// TwinCAT 3 PLC project ControlPanel
// ProgramVersion: 3.1.4024.0
// libraries:
//   Tc2_HVAC, * (Beckhoff Automation GmbH)
//   Tc2_ModbusSrv, * (Beckhoff Automation GmbH)
//   Tc2_Standard, * (Beckhoff Automation GmbH)
//   Tc2_System, * (Beckhoff Automation GmbH)
//   Tc3_Module, * (Beckhoff Automation GmbH)
// project tree:
//   DUTs/ FactoryIO_Input.TcDUT, FactoryIO_Output.TcDUT
//   GVLs/ GVL.TcGVL, GVL_System.TcGVL
//   / PlcTask.TcTTO
//   POUs/ Blink.TcPOU, ControlPanel.TcPOU, MAIN.TcPOU, MyBlink.TcPOU, ReadModbusCoils.TcPOU, ReadModbusReg.TcPOU
// real-time tasks:
//   TASK PlcTask: cycle T#10ms, priority 20, ADS port 350

CONFIGURATION ControlPanel
    RESOURCE PLC ON TwinCAT3
        TASK PlcTask(INTERVAL := T#10ms, PRIORITY := 20);
        PROGRAM MAIN WITH PlcTask : MAIN;
    END_RESOURCE
END_CONFIGURATION

// ---- DUTs/FactoryIO_Input.TcDUT
TYPE FactoryIO_Input :
STRUCT
	bAtBufferEntry	:	BOOL;
	bAtBufferExit	:	BOOL;
	bAtExit			:	BOOL;
	bStartButton	: 	BOOL;
	bResetButton	: 	BOOL;
	bStopButton		: 	BOOL;
	bAuto			: 	BOOL;
	bEmgStop		: 	BOOL;
	bManual			: 	BOOL;
	nSpeed			:	WORD;
END_STRUCT
END_TYPE

// ---- DUTs/FactoryIO_Output.TcDUT
TYPE FactoryIO_Output :
STRUCT
	bStopBlade		:	BOOL;
	bStartLight		:	BOOL;
	bResetLight		:	BOOL;
	bStopLight		:	BOOL;
	nBufferConveyor	: 	WORD;
	nExitConveyor	: 	WORD;
	nCounter		:	WORD;
END_STRUCT
END_TYPE

// ---- GVLs/GVL.TcGVL
{attribute 'qualified_only'}
VAR_GLOBAL
	// Digital IO in FactoryIO Outputs
	mb_Input_Coils		:	ARRAY [0..3] OF BOOL;
	// Digital IO in FactoryIO Inputs
	mb_Output_Coils		:   ARRAY [0..9] OF BOOL;
	// Analog IO in FactoryIO Outputs
	mb_Input_Registers	: 	ARRAY [0..2] OF WORD;
	// Analog IO in FactoryIO Inputs
	mb_Output_Registers	: 	ARRAY [0..1] OF WORD;
	
	nState				: INT;
END_VAR

// ---- GVLs/GVL_System.TcGVL
{attribute 'qualified_only'}
VAR_GLOBAL
	isResetON	: BOOL;
	isStopON	: BOOL;
	isEmgStopON	: BOOL;
	
END_VAR

// ---- POUs/MAIN.TcPOU
PROGRAM MAIN
VAR
	(*
	fbReadRegs        : FB_MBReadRegs;
    bReadRegs         : BOOL;
    bReadRegsBusy     : BOOL;
    bReadRegsError    : BOOL;
    nReadRegsErrorId  : UDINT;
    nReadRegsCount    : UDINT;
    nQuantity         : WORD:=2;
    nMBAddr           : WORD:=24;
    arrData           : ARRAY [1..2] OF WORD;
	*)
	
	//myBlink	: Array[0..7] OF MyBlink();
	redBlink	: MyBlink();
	yellowBlink	: MyBlink();
	greenBlink	: MyBlink();
	controlPanel 	:	ControlPanel();
	
END_VAR

Blink();


ControlPanel();

END_PROGRAM

// ---- POUs/MyBlink.TcPOU
FUNCTION_BLOCK MyBlink
VAR_INPUT
	tBlinkTime			: TON;
	bEnable				: BOOL;
	bBlinkHz			: BOOL;
	tTimeOn				: TIME := T#2S;
	tTimeOff 			: TIME := tTimeOn/2;
END_VAR
VAR_OUTPUT
	bBlink				: BOOL;
END_VAR
VAR
END_VAR

// SET Timer ON
tBlinkTime(IN:=NOT tBlinkTime.Q, PT:= tTimeON);

// Set Timer OFF
bBlinkHz := tBlinkTime.ET >= tTimeOff;

// OUTPUT
bBlink := bBlinkHz AND bEnable;

END_FUNCTION_BLOCK

// ---- POUs/ControlPanel.TcPOU
FUNCTION_BLOCK ControlPanel
VAR_INPUT
	
	
END_VAR
VAR_OUTPUT
	
END_VAR
VAR
	isResetON	: BOOL;
	isStopON	: BOOL;
	isEmgStopON	: BOOL;
	isSystemON	: BOOL;
	
	factoryIO_Input	: FactoryIO_Input;
	i	: INT;
	
	(*
	bAtBufferEntry	:	BOOL;
	bAtBufferExit	:	BOOL;
	bAtExit			:	BOOL;
	bStartButton	: 	BOOL;
	bResetButton	: 	BOOL;
	bStopButton		: 	BOOL;
	bAuto			: 	BOOL;
	bEmgStop		: 	BOOL;
	bManual			: 	BOOL;
	*)
	
	blink			: MyBlink();
END_VAR

{region "READ Values from Sensors"}
	(*
	bAtBufferEntry	:=	GVL.mb_Output_Coils[0];
	bAtBufferExit	:= 	GVL.mb_Output_Coils[1];
	bAtExit			:=	GVL.mb_Output_Coils[2];
	bStartButton	:=	GVL.mb_Output_Coils[3];
	bResetButton	:= 	GVL.mb_Output_Coils[4];
	bStopButton		:= 	GVL.mb_Output_Coils[5];
	bAuto			:=	GVL.mb_Output_Coils[6];
	bEmgStop	 	:= 	GVL.mb_Output_Coils[7];
	bManual	 		:= 	GVL.mb_Output_Coils[8];
	*)
	 
	factoryIO_Input.bAtBufferEntry	:=	GVL.mb_Output_Coils[0];
	factoryIO_Input.bAtBufferExit	:=	GVL.mb_Output_Coils[1];
	factoryIO_Input.bAtExit			:=	GVL.mb_Output_Coils[2];
	factoryIO_Input.bStartButton	:=	GVL.mb_Output_Coils[3];
	factoryIO_Input.bResetButton	:=	GVL.mb_Output_Coils[4];
	factoryIO_Input.bStopButton		:=	GVL.mb_Output_Coils[5];
	factoryIO_Input.bAuto			:=	GVL.mb_Output_Coils[6];
	factoryIO_Input.bEmgStop		:=	GVL.mb_Output_Coils[7];
	factoryIO_Input.bManual			:=	GVL.mb_Output_Coils[8];
	factoryIO_Input.nSpeed			:=	GVL.mb_Output_Registers[0];
		 
	
	isEmgStopON	:=	GVL_System.isEmgStopON;
	isResetON 	:= 	GVL_System.isResetON;
	isStopON	:= 	GVL_System.isStopON;
	isSystemON	:= 	GVL_System.isSystemON;	
{endregion}
	 
	 
{region "LOGIC"}
	{REGION "Memory BIT FOR SystemON"}
		// When isSystemON memory bit is true system is ready to run
		IF isResetON OR isStopON THEN
			IF isEmgStopON AND factoryIO_Input.bStartButton THEN
				isSystemON := TRUE;
			END_IF;
		END_IF;
		
		IF NOT isEmgStopON OR NOT factoryIO_Input.bStopButton THEN
			isSystemON := FALSE;
		END_IF;		
	{endregion}

	{REGION "Memory Bit FOR isEmgStopON - Set/Reset"}
		IF factoryIO_Input.bEmgStop THEN
			isEmgStopON := TRUE;
		END_IF;
		
		IF NOT factoryIO_Input.bEmgStop THEN
			isEmgStopON := FALSE;
		END_IF;
	{endregion}
	
	{REGION "Memory Bit FOR isResetON - Set/Reset"}
		IF factoryIO_Input.bResetButton AND isEmgStopON AND NOT isStopON THEN
			isResetON := TRUE;
		END_IF;
		
		IF factoryIO_Input.bStartButton THEN
			isResetON := FALSE;
		END_IF;		
	{endregion}

	{REGION "Memory Bit FOR isStopON - Set/Reset"}		 
		IF NOT factoryIO_Input.bStopButton AND isEmgStopON THEN
			isStopON := TRUE;
		END_IF;
		
		IF isSystemON OR NOT isEmgStopON THEN
			isStopON := FALSE;
		END_IF;
		
	{endregion}

	// ======= OUTPUTS =========
	
	{REGION Start Light ON with Coil (Assignment)}
		GVL.mb_Input_Coils[1] := isSystemON OR ((isResetON OR (NOT isResetON AND isStopON)) AND isEmgStopON AND NOT isSystemON AND blink);
	{endregion}
			  
	{REGION Reset Light ON with Coil (Assignment)}	 
		GVL.mb_Input_Coils[2] := (isResetON OR (NOT isResetON AND blink)) AND isEmgStopON AND NOT isStopON AND NOT isSystemON;
	{endregion}
	
	{REGION Stop Light ON with Coil (Assignment)}
		GVL.mb_Input_Coils[3] := (isEmgStopON OR isStopON OR (NOT isEmgStopON AND blink)) AND NOT isSystemON;
	{endregion}

	
	GVL_System.isEmgStopON:= isEmgStopON;
	GVL_System.isResetON:= isResetON;
	GVL_System.isStopON:= isStopON;
	GVL_System.isSystemON := isSystemON;
	
{endregion}

END_FUNCTION_BLOCK

// ---- POUs/Blink.TcPOU
PROGRAM Blink
VAR
	hvacBlink 	: FB_HVACBlink();
	bEnable		: BOOL;
	tTimeOn		: TIME := T#2S;
	tTimeOff 	: TIME := T#1S;
END_VAR

VAR_OUTPUT
	bBlink			: BOOL;
	tNextSwitching  :TIME;
END_VAR

hvacBlink(bEnable:=bEnable,
tTimeOn:=tTimeOn,
tTimeOff:=tTimeOff,
bBlink=>,
tNextSwitching=>);

END_PROGRAM

// ---- POUs/ReadModbusCoils.TcPOU
PROGRAM ReadModbusCoils
VAR
	fbReadCoils       : FB_MBReadCoils;
    bReadCoils        : BOOL;
    bReadCoilsBusy    : BOOL;
    bReadCoilsError   : BOOL;
    nReadCoilsErrorId : UDINT;
    nReadCoilsCount   : UDINT;
    nQuantity         : WORD := 10;
    nMBAddr           : WORD := 32768;
    arrData           : ARRAY [0..1] OF BYTE;
	nTCPPort		  : UINT 	:= 502;
	nUnitID			  : BYTE	:= 255;
	tTimeout		  : TIME	:= T#1S;
END_VAR

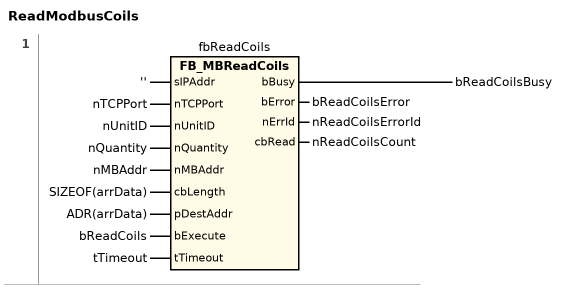
// NETWORK 1
fbReadCoils(
    sIPAddr := '',
    nTCPPort := nTCPPort,
    nUnitID := nUnitID,
    nQuantity := nQuantity,
    nMBAddr := nMBAddr,
    cbLength := SIZEOF(arrData),
    pDestAddr := ADR(arrData),
    bExecute := bReadCoils,
    tTimeout := tTimeout,
    bError => bReadCoilsError,
    nErrId => nReadCoilsErrorId,
    cbRead => nReadCoilsCount); // FB_MBReadCoils
bReadCoilsBusy := fbReadCoils.bBusy;

END_PROGRAM

// ---- POUs/ReadModbusReg.TcPOU
PROGRAM ReadModbusReg
VAR
	fbReadRegs        : FB_MBReadRegs;
    bReadRegs         : BOOL;
    bReadRegsBusy     : BOOL;
    bReadRegsError    : BOOL;
    nReadRegsErrorId  : UDINT;
    nReadRegsCount    : UDINT;
    nQuantity         : WORD:=2;
    nMBAddr           : WORD:=32768;
    arrData           : ARRAY [0..1] OF WORD;
	nTCPPort		  : UINT	:= 502;
	nUnitID			  : BYTE	:= 255;
	tTimeout		  : TIME	:= T#1S;
END_VAR

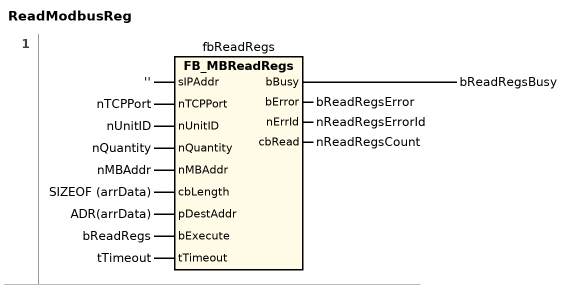
// NETWORK 1
fbReadRegs(
    sIPAddr := '',
    nTCPPort := nTCPPort,
    nUnitID := nUnitID,
    nQuantity := nQuantity,
    nMBAddr := nMBAddr,
    cbLength := SIZEOF (arrData),
    pDestAddr := ADR(arrData),
    bExecute := bReadRegs,
    tTimeout := tTimeout,
    bError => bReadRegsError,
    nErrId => nReadRegsErrorId,
    cbRead => nReadRegsCount); // FB_MBReadRegs
bReadRegsBusy := fbReadRegs.bBusy;

END_PROGRAM
